// TwinCAT 3 PLC project TRAJ_ADS_SERVER
// ProgramVersion: 3.1.4020.4
// libraries:
//   Tc2_ControllerToolbox, * (Beckhoff Automation GmbH)
//   Tc2_Standard, * (Beckhoff Automation GmbH)
//   Tc2_System, * (Beckhoff Automation GmbH)
//   Tc3_Interfaces, * (Beckhoff Automation GmbH)
//   Tc3_Module, * (Beckhoff Automation GmbH)
// project tree:
//   DUTs/ ROBOT_STATUS.TcDUT, TRAJECTORY.TcDUT, TRAJ_POINT.TcDUT
//   GVLs/ CONST.TcGVL
//   / PlcTask.TcTTO
//   POUs/ MAIN.TcPOU
// real-time tasks:
//   TASK PlcTask: cycle T#10ms, priority 6, ADS port 350
// motion (NC):
//   TASK NC-Task 1 SAF: cycle T#2ms, priority 4, ADS port 501
//   TASK NC-Task 1 SVB: cycle T#10ms, priority 8, ADS port 511
//   AXIS Axis 1 (id 1)
//     OtherSettings: AllowMotionCmdToSlave=true
//     encoder EncType=19
//       EncPara: MaxCount=#xffffffff
//     drive DrvType=16
//       DrvPara: MaxCount=#xffffffff, DriveControlDWord=#x00000100
//         Analog: ScaleFactorActTorque=0.1
//         TimeComp: TaskDelayCycles=1
//     controller CtrType=1
//       CtrPara: PriorControlFactor=1
//         Observer: BandWidth=20

CONFIGURATION TRAJ_ADS_SERVER
    RESOURCE PLC ON TwinCAT3
        TASK PlcTask(INTERVAL := T#10ms, PRIORITY := 6);
        PROGRAM MAIN WITH PlcTask : MAIN;
    END_RESOURCE
END_CONFIGURATION

// ---- DUTs/ROBOT_STATUS.TcDUT
TYPE ROBOT_STATUS :
STRUCT
		driverPowered: BYTE:=CONST.ROBO_STATUS_TRUE; //驱动是否上电
		eStopped:  BYTE:=CONST.ROBO_STATUS_FALSE; //是否非正常停止(如碰撞)
		inError: BYTE:=CONST.ROBO_STATUS_FALSE; //是否发生错误
		inMotion:BYTE:=CONST.ROBO_STATUS_TRUE; //是否在运动
		motionPossible :BYTE:=CONST.ROBO_STATUS_TRUE; //是否可以运动
		mode: BYTE:=CONST.ROBO_MODE_AUTO; //当前的模式 自动/手动/未知
		errorCode: UINT:=CONST.ROBO_ERRORCODE_NONE;   //错误码：自定义
		position        :TRAJ_POINT;   //采集的关节位置
END_STRUCT

END_TYPE

// ---- DUTs/TRAJECTORY.TcDUT
TYPE TRAJECTORY :
STRUCT
		cmd           :UINT:=CONST.TRAJ_CMD_STOP;                           //命令
	    step          :UINT:=1;                        //轨迹点的时间间隔，默认1ms
		size     	  :UDINT:=0;                          //轨迹点的数目
		index         :UDINT:=0;                          //当前轨迹点的起始index
		points        :ARRAY[1..CONST.PTS_NUMBER] OF TRAJ_POINT;   //要执行的一系列轨迹点  
END_STRUCT
END_TYPE

// ---- DUTs/TRAJ_POINT.TcDUT
TYPE TRAJ_POINT :
STRUCT
	joints    : ARRAY [0..6] OF REAL;              //关节的位置数据(7关节)
END_STRUCT
END_TYPE

// ---- GVLs/CONST.TcGVL
{attribute 'qualified_only'}
VAR_GLOBAL CONSTANT
	  PTS_NUMBER:UDINT:=100000;   //轨迹点的数目
	
	//轨迹命令
	 TRAJ_CMD_NEW:BYTE :=  1;  //读入轨迹
	 TRAJ_CMD_START:BYTE :=  2;  //开始运动
	 TRAJ_CMD_PAUSE:BYTE :=  3;  //暂停运动
	 TRAJ_CMD_STOP:BYTE :=  0;  //停止
	
	
	//机器人模式
	 ROBO_MODE_AUTO:   BYTE :=  1; //自动模式
	 ROBO_MODE_MANNUL:   BYTE :=  2;//手动模式
	 ROBO_MODE_UNKNOW:   BYTE :=  3;//未知模式
	 
	 
	 //状态，True或者FALSE
	 ROBO_STATUS_TRUE:BYTE:=255;
	 ROBO_STATUS_FALSE:BYTE:=0;
	 
	 //错误码
	 ROBO_ERRORCODE_NONE:UINT:=0; //无错误
	 ROBO_ERRORCODE_ALARM:UINT:=10; //报警错误
	 

END_VAR

// ---- POUs/MAIN.TcPOU
PROGRAM MAIN

VAR
	//VREP 控制数据
	traj_cmd                :UINT:=CONST.TRAJ_CMD_STOP; //命令
	traj_step               :UINT:=1;//轨迹的步长
	traj_size               :UDINT:=0;            //轨迹点的个数
	traj_index              :UDINT:=0;
	traj_path               :TRAJECTORY; //轨迹路径点：固定10000个点，间隔1ms(上位机指定)
	
	//机器人状态反馈
	robo_status            :ROBOT_STATUS;
	
	j: INT;
END_VAR



//上报机器人状态和关节位置()
SEND_ROBOT_STATUS();


//每个循环读取指令和轨迹点
traj_cmd:=traj_path.cmd;   //控制命令CMD


CASE traj_cmd OF
CONST.TRAJ_CMD_NEW:   //初始化：读取变量然后将原来的cmd改为START(或PAUSE)
	//traj_index和traj_step只会在此处读取！
	traj_size:=traj_path.size; 
	traj_index:=traj_path.index; 
	traj_step:=traj_path.step;  //步长1ms默认
	traj_path.cmd:=CONST.TRAJ_CMD_PAUSE;  //修改traj_path为PAUSE

	FUNC_NEW(); //接口实现:新路径
CONST.TRAJ_CMD_START:
	IF traj_index>=traj_size THEN
		traj_cmd:=CONST.TRAJ_CMD_STOP;
	END_IF
	robo_status.inMotion:=CONST.ROBO_STATUS_TRUE;//正在运动
	traj_index:=traj_index+1;
	FOR j:=1 TO 7 BY 1 DO
	   //traj_path.points[traj_index].joints[j]:轨迹点1的关节J的数据
	END_FOR
	FUNC_START(); //接口实现:开始运动
CONST.TRAJ_CMD_STOP:    
	traj_size:=0;
	traj_index:=0;
	traj_path.cmd:=CONST.TRAJ_CMD_PAUSE;  //设置为STOP  
	robo_status.inMotion:=CONST.ROBO_STATUS_FALSE;//停止运动
	FUNC_PAUSE(); //接口实现:停止运动
ELSE
	//暂停时不改变size和index
	robo_status.inMotion:=CONST.ROBO_STATUS_FALSE;//停止运动
	FUNC_PAUSE(); //接口实现:暂停运行哦那个
END_CASE;

METHOD FUNC_NEW : BOOL
VAR_INPUT
END_VAR
FUNC_NEW:=TRUE;
END_METHOD

METHOD FUNC_PAUSE : BOOL
VAR_INPUT
END_VAR
FUNC_PAUSE:=TRUE;
END_METHOD

METHOD FUNC_START : BOOL
VAR_INPUT
END_VAR
FUNC_START:=TRUE;
END_METHOD

METHOD FUNC_STOP : BOOL
VAR_INPUT
END_VAR
FUNC_STOP:=TRUE;
END_METHOD

METHOD SEND_ROBOT_STATUS : BOOL
VAR_INPUT
END_VAR
robo_status.driverPowered:=CONST.ROBO_STATUS_TRUE;//驱动上电
robo_status.eStopped:=CONST.ROBO_STATUS_FALSE;//未意外停止
robo_status.inError:=CONST.ROBO_STATUS_FALSE;//未发生错误
//robo_status.inMotion:=CONST.ROBO_STATUS_FALSE;//正在运动
robo_status.motionPossible:=CONST.ROBO_STATUS_TRUE;//可以运动
robo_status.errorCode:=CONST.ROBO_ERRORCODE_NONE;//错误码


//关节位置:从私服驱动中读取
robo_status.position.joints[0]:=SIN(traj_index*0.0001)+1.0;
robo_status.position.joints[1]:=SIN(traj_index*0.0001)+2.0;
robo_status.position.joints[2]:=SIN(traj_index*0.0001)+3.0;
robo_status.position.joints[3]:=SIN(traj_index*0.0001)+4.0;
robo_status.position.joints[4]:=SIN(traj_index*0.0001)+5.0;
robo_status.position.joints[5]:=SIN(traj_index*0.0001)+6.0;
robo_status.position.joints[6]:=SIN(traj_index*0.0001)+7.0;


SEND_ROBOT_STATUS:=TRUE;
END_METHOD

END_PROGRAM
